TYPE ST_Event :
STRUCT
	What_happend			: STRING[20];
	sEventText				: STRING[255];
	eEventType				: E_EventType;
	eEventSeverity			: TcEventSeverity;
	dtTimeStamp				: DATE_AND_TIME;
END_STRUCT
END_TYPE

(* stored: Version 1.1.0.1, ProductVersion 3.1.4024.12
   DUT ST_Event: Id {965e98fa-4f80-4075-b883-64e0c73472b0} *)
